VISUALIZATION View_3Lifts  // 2x2
END_VISUALIZATION

(* stored: Version 1.1.0.1
   Visu View_3Lifts: Id {27ebe13a-22b5-4039-95de-4cf24d858fd9} *)
